PROGRAM MAIN
VAR
END_VAR

Control_Panel_Sequencer();

END_PROGRAM

(* stored: Version 1.1.0.1, ProductVersion 3.1.4024.15
   POU MAIN: Id {e1885f29-6855-4a0a-b957-883197d57311}, SpecialFunc None *)
